// TIA Portal V16 export
// export: Created 2024-05-11T02:56:22.535184Z, ExportSetting WithDefaults, DisplayName Totally Integrated Automation Portal, DisplayVersion V16, DisplayName TIA Portal Version Control Interface, DisplayVersion V16, DisplayName TIA Portal Openness, DisplayVersion V16, DisplayName STEP 7 Professional, DisplayVersion V16, DisplayName STEP 7 Safety, DisplayVersion V16, DisplayName WinCC Professional, DisplayVersion V16
FUNCTION_BLOCK "K11_入口自动"   // FB11, LAD
{ S7_Optimized_Access := 'TRUE' }
VERSION : 0.1
// stored: AutoNumber false, IsIECCheckEnabled false, IsRetainMemResEnabled false, MemoryReserve 100, SetENOAutomatically false, UDAEnableTagReadback false
   VAR_TEMP
      EN_提升机上升指令 : Array[1..8] of Bool;
      EN_提升机下降指令 : Array[1..8] of Bool;
      EN_阻挡上升指令 : Array[1..8] of Bool;
      EN_阻挡下降指令 : Array[1..8] of Bool;
   END_VAR
   VAR_TEMP   // added for the SCL form of the ladder/FBD networks
      _w1 : Bool;
   END_VAR
BEGIN

REGION Network 1: @SN1=入口部
END_REGION

REGION Network 2: @选择分支
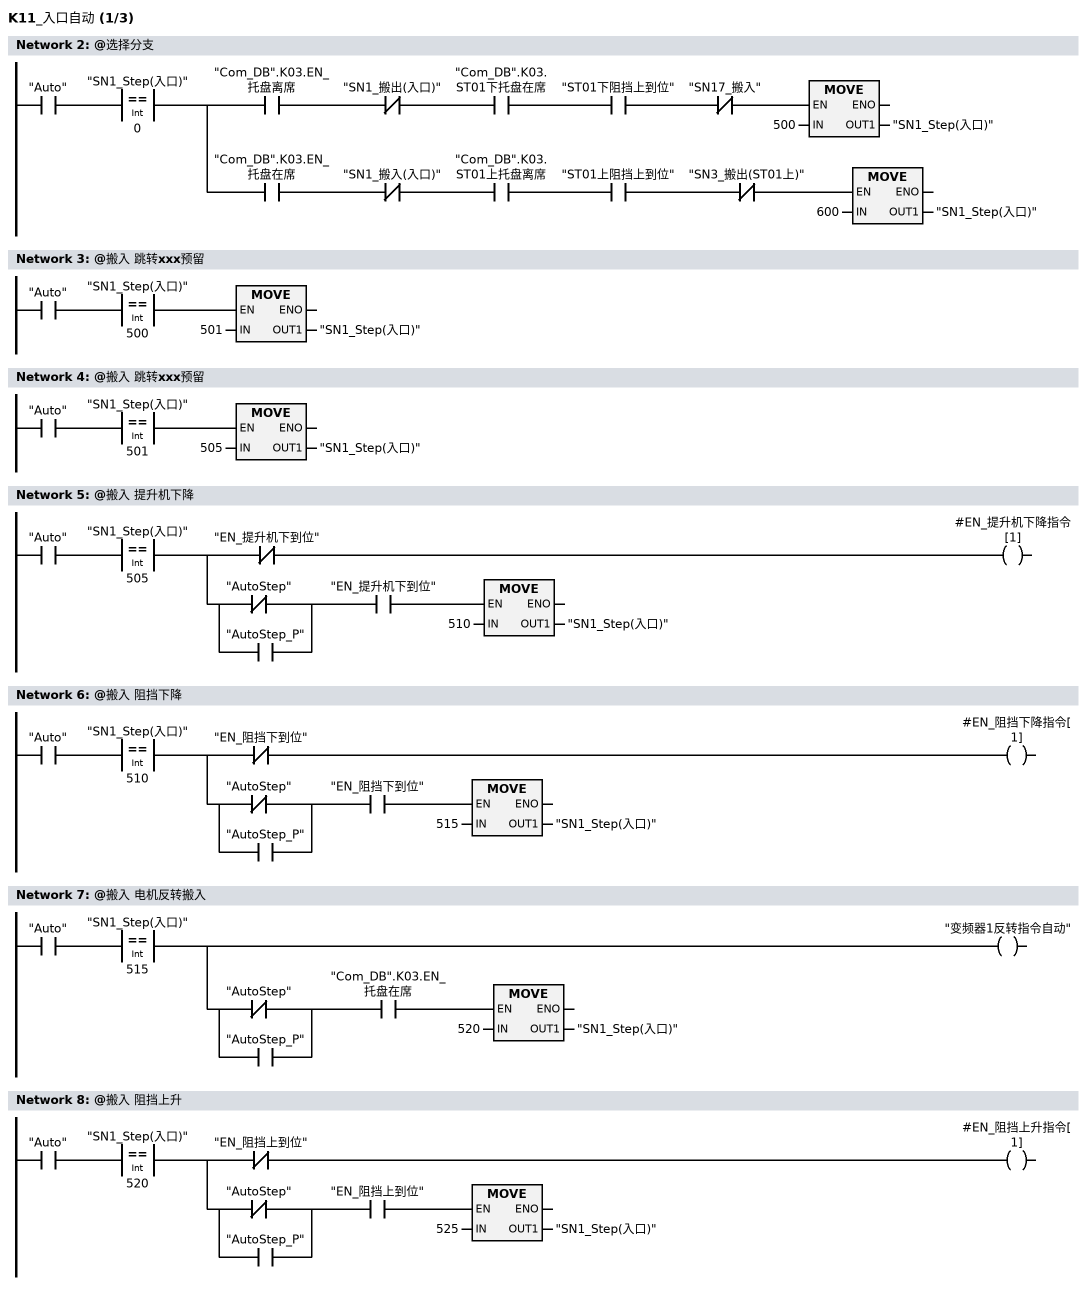
   RUNG wire#powerrail
      Contact( "Auto" )
      { S7_Templates := "SrcType := Int" } EQ_Contact(in1 := "SN1_Step(入口)", in2 := 0)
      wire#w1
      Contact( "Com_DB".K03.EN_托盘离席 )
      I_Contact( "SN1_搬出(入口)" )
      Contact( "Com_DB".K03.ST01下托盘在席 )
      Contact( "ST01下阻挡上到位" )
      I_Contact( "SN17_搬入" )
      Move(in := 500, out1 => "SN1_Step(入口)")
   END_RUNG
   RUNG wire#w1
      Contact( "Com_DB".K03.EN_托盘在席 )
      I_Contact( "SN1_搬入(入口)" )
      Contact( "Com_DB".K03.ST01上托盘离席 )
      Contact( "ST01上阻挡上到位" )
      I_Contact( "SN3_搬出(ST01上)" )
      Move(in := 600, out1 => "SN1_Step(入口)")
   END_RUNG
   // the same network as SCL:
   #_w1 := "Auto" AND ("SN1_Step(入口)" = 0);
   IF #_w1 AND "Com_DB".K03.EN_托盘离席 AND NOT "SN1_搬出(入口)" AND "Com_DB".K03.ST01下托盘在席 AND "ST01下阻挡上到位" AND NOT "SN17_搬入" THEN
       "SN1_Step(入口)" := 500;
   END_IF;
   IF #_w1 AND "Com_DB".K03.EN_托盘在席 AND NOT "SN1_搬入(入口)" AND "Com_DB".K03.ST01上托盘离席 AND "ST01上阻挡上到位" AND NOT "SN3_搬出(ST01上)" THEN
       "SN1_Step(入口)" := 600;
   END_IF;
END_REGION

REGION Network 3: @搬入 跳转xxx预留
   RUNG wire#powerrail
      Contact( "Auto" )
      { S7_Templates := "SrcType := Int" } EQ_Contact(in1 := "SN1_Step(入口)", in2 := 500)
      Move(in := 501, out1 => "SN1_Step(入口)")
   END_RUNG
   // the same network as SCL:
   IF "Auto" AND ("SN1_Step(入口)" = 500) THEN "SN1_Step(入口)" := 501; END_IF;
END_REGION

REGION Network 4: @搬入 跳转xxx预留
   RUNG wire#powerrail
      Contact( "Auto" )
      { S7_Templates := "SrcType := Int" } EQ_Contact(in1 := "SN1_Step(入口)", in2 := 501)
      Move(in := 505, out1 => "SN1_Step(入口)")
   END_RUNG
   // the same network as SCL:
   IF "Auto" AND ("SN1_Step(入口)" = 501) THEN "SN1_Step(入口)" := 505; END_IF;
END_REGION

REGION Network 5: @搬入 提升机下降
   RUNG wire#powerrail
      Contact( "Auto" )
      { S7_Templates := "SrcType := Int" } EQ_Contact(in1 := "SN1_Step(入口)", in2 := 505)
      wire#w1
      I_Contact( "EN_提升机下到位" )
      Coil( #EN_提升机下降指令[1] )
   END_RUNG
   RUNG wire#w1
      I_Contact( "AutoStep" )
      wire#w2
      Contact( "EN_提升机下到位" )
      Move(in := 510, out1 => "SN1_Step(入口)")
   END_RUNG
   RUNG wire#w1
      Contact( "AutoStep_P" )
   END_RUNG wire#w2
   // the same network as SCL:
   #_w1 := "Auto" AND ("SN1_Step(入口)" = 505);
   #EN_提升机下降指令[1] := #_w1 AND NOT "EN_提升机下到位";
   IF #_w1 AND (NOT "AutoStep" OR "AutoStep_P") AND "EN_提升机下到位" THEN "SN1_Step(入口)" := 510; END_IF;
END_REGION

REGION Network 6: @搬入 阻挡下降
   RUNG wire#powerrail
      Contact( "Auto" )
      { S7_Templates := "SrcType := Int" } EQ_Contact(in1 := "SN1_Step(入口)", in2 := 510)
      wire#w1
      I_Contact( "EN_阻挡下到位" )
      Coil( #EN_阻挡下降指令[1] )
   END_RUNG
   RUNG wire#w1
      I_Contact( "AutoStep" )
      wire#w2
      Contact( "EN_阻挡下到位" )
      Move(in := 515, out1 => "SN1_Step(入口)")
   END_RUNG
   RUNG wire#w1
      Contact( "AutoStep_P" )
   END_RUNG wire#w2
   // the same network as SCL:
   #_w1 := "Auto" AND ("SN1_Step(入口)" = 510);
   #EN_阻挡下降指令[1] := #_w1 AND NOT "EN_阻挡下到位";
   IF #_w1 AND (NOT "AutoStep" OR "AutoStep_P") AND "EN_阻挡下到位" THEN "SN1_Step(入口)" := 515; END_IF;
END_REGION

REGION Network 7: @搬入 电机反转搬入
   RUNG wire#powerrail
      Contact( "Auto" )
      { S7_Templates := "SrcType := Int" } EQ_Contact(in1 := "SN1_Step(入口)", in2 := 515)
      wire#w1
      Coil( "变频器1反转指令自动" )
   END_RUNG
   RUNG wire#w1
      I_Contact( "AutoStep" )
      wire#w2
      Contact( "Com_DB".K03.EN_托盘在席 )
      Move(in := 520, out1 => "SN1_Step(入口)")
   END_RUNG
   RUNG wire#w1
      Contact( "AutoStep_P" )
   END_RUNG wire#w2
   // the same network as SCL:
   "变频器1反转指令自动" := "Auto" AND ("SN1_Step(入口)" = 515);
   IF "变频器1反转指令自动" AND (NOT "AutoStep" OR "AutoStep_P") AND "Com_DB".K03.EN_托盘在席 THEN
       "SN1_Step(入口)" := 520;
   END_IF;
END_REGION

REGION Network 8: @搬入 阻挡上升
   RUNG wire#powerrail
      Contact( "Auto" )
      { S7_Templates := "SrcType := Int" } EQ_Contact(in1 := "SN1_Step(入口)", in2 := 520)
      wire#w1
      I_Contact( "EN_阻挡上到位" )
      Coil( #EN_阻挡上升指令[1] )
   END_RUNG
   RUNG wire#w1
      I_Contact( "AutoStep" )
      wire#w2
      Contact( "EN_阻挡上到位" )
      Move(in := 525, out1 => "SN1_Step(入口)")
   END_RUNG
   RUNG wire#w1
      Contact( "AutoStep_P" )
   END_RUNG wire#w2
   // the same network as SCL:
   #_w1 := "Auto" AND ("SN1_Step(入口)" = 520);
   #EN_阻挡上升指令[1] := #_w1 AND NOT "EN_阻挡上到位";
   IF #_w1 AND (NOT "AutoStep" OR "AutoStep_P") AND "EN_阻挡上到位" THEN "SN1_Step(入口)" := 525; END_IF;
END_REGION

REGION Network 9: @等搬入标志清除
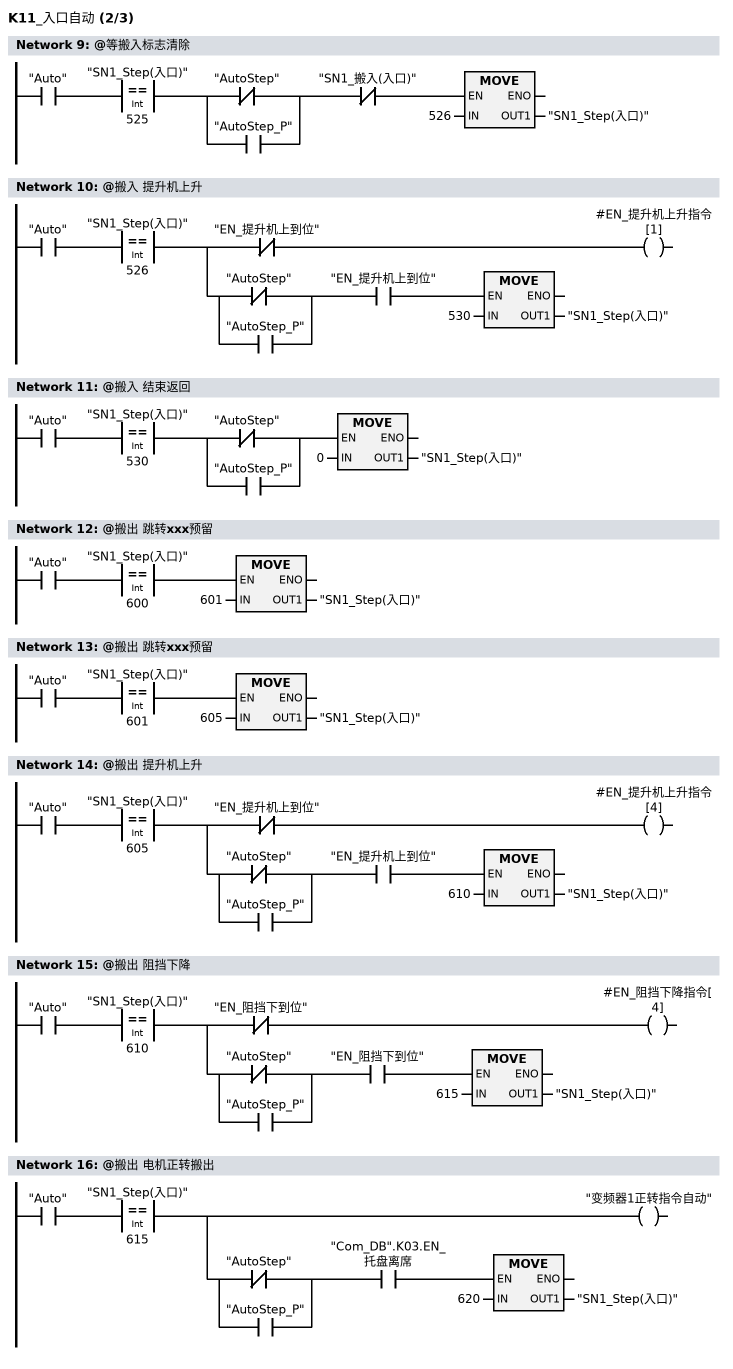
   RUNG wire#powerrail
      Contact( "Auto" )
      { S7_Templates := "SrcType := Int" } EQ_Contact(in1 := "SN1_Step(入口)", in2 := 525)
      wire#w1
      I_Contact( "AutoStep" )
      wire#w2
      I_Contact( "SN1_搬入(入口)" )
      Move(in := 526, out1 => "SN1_Step(入口)")
   END_RUNG
   RUNG wire#w1
      Contact( "AutoStep_P" )
   END_RUNG wire#w2
   // the same network as SCL:
   IF "Auto" AND ("SN1_Step(入口)" = 525) AND (NOT "AutoStep" OR "AutoStep_P") AND NOT "SN1_搬入(入口)" THEN
       "SN1_Step(入口)" := 526;
   END_IF;
END_REGION

REGION Network 10: @搬入 提升机上升
   RUNG wire#powerrail
      Contact( "Auto" )
      { S7_Templates := "SrcType := Int" } EQ_Contact(in1 := "SN1_Step(入口)", in2 := 526)
      wire#w1
      I_Contact( "EN_提升机上到位" )
      Coil( #EN_提升机上升指令[1] )
   END_RUNG
   RUNG wire#w1
      I_Contact( "AutoStep" )
      wire#w2
      Contact( "EN_提升机上到位" )
      Move(in := 530, out1 => "SN1_Step(入口)")
   END_RUNG
   RUNG wire#w1
      Contact( "AutoStep_P" )
   END_RUNG wire#w2
   // the same network as SCL:
   #_w1 := "Auto" AND ("SN1_Step(入口)" = 526);
   #EN_提升机上升指令[1] := #_w1 AND NOT "EN_提升机上到位";
   IF #_w1 AND (NOT "AutoStep" OR "AutoStep_P") AND "EN_提升机上到位" THEN "SN1_Step(入口)" := 530; END_IF;
END_REGION

REGION Network 11: @搬入 结束返回
   RUNG wire#powerrail
      Contact( "Auto" )
      { S7_Templates := "SrcType := Int" } EQ_Contact(in1 := "SN1_Step(入口)", in2 := 530)
      wire#w1
      I_Contact( "AutoStep" )
      wire#w2
      Move(in := 0, out1 => "SN1_Step(入口)")
   END_RUNG
   RUNG wire#w1
      Contact( "AutoStep_P" )
   END_RUNG wire#w2
   // the same network as SCL:
   IF "Auto" AND ("SN1_Step(入口)" = 530) AND (NOT "AutoStep" OR "AutoStep_P") THEN
       "SN1_Step(入口)" := 0;
   END_IF;
END_REGION

REGION Network 12: @搬出 跳转xxx预留
   RUNG wire#powerrail
      Contact( "Auto" )
      { S7_Templates := "SrcType := Int" } EQ_Contact(in1 := "SN1_Step(入口)", in2 := 600)
      Move(in := 601, out1 => "SN1_Step(入口)")
   END_RUNG
   // the same network as SCL:
   IF "Auto" AND ("SN1_Step(入口)" = 600) THEN "SN1_Step(入口)" := 601; END_IF;
END_REGION

REGION Network 13: @搬出 跳转xxx预留
   RUNG wire#powerrail
      Contact( "Auto" )
      { S7_Templates := "SrcType := Int" } EQ_Contact(in1 := "SN1_Step(入口)", in2 := 601)
      Move(in := 605, out1 => "SN1_Step(入口)")
   END_RUNG
   // the same network as SCL:
   IF "Auto" AND ("SN1_Step(入口)" = 601) THEN "SN1_Step(入口)" := 605; END_IF;
END_REGION

REGION Network 14: @搬出 提升机上升
   RUNG wire#powerrail
      Contact( "Auto" )
      { S7_Templates := "SrcType := Int" } EQ_Contact(in1 := "SN1_Step(入口)", in2 := 605)
      wire#w1
      I_Contact( "EN_提升机上到位" )
      Coil( #EN_提升机上升指令[4] )
   END_RUNG
   RUNG wire#w1
      I_Contact( "AutoStep" )
      wire#w2
      Contact( "EN_提升机上到位" )
      Move(in := 610, out1 => "SN1_Step(入口)")
   END_RUNG
   RUNG wire#w1
      Contact( "AutoStep_P" )
   END_RUNG wire#w2
   // the same network as SCL:
   #_w1 := "Auto" AND ("SN1_Step(入口)" = 605);
   #EN_提升机上升指令[4] := #_w1 AND NOT "EN_提升机上到位";
   IF #_w1 AND (NOT "AutoStep" OR "AutoStep_P") AND "EN_提升机上到位" THEN "SN1_Step(入口)" := 610; END_IF;
END_REGION

REGION Network 15: @搬出 阻挡下降
   RUNG wire#powerrail
      Contact( "Auto" )
      { S7_Templates := "SrcType := Int" } EQ_Contact(in1 := "SN1_Step(入口)", in2 := 610)
      wire#w1
      I_Contact( "EN_阻挡下到位" )
      Coil( #EN_阻挡下降指令[4] )
   END_RUNG
   RUNG wire#w1
      I_Contact( "AutoStep" )
      wire#w2
      Contact( "EN_阻挡下到位" )
      Move(in := 615, out1 => "SN1_Step(入口)")
   END_RUNG
   RUNG wire#w1
      Contact( "AutoStep_P" )
   END_RUNG wire#w2
   // the same network as SCL:
   #_w1 := "Auto" AND ("SN1_Step(入口)" = 610);
   #EN_阻挡下降指令[4] := #_w1 AND NOT "EN_阻挡下到位";
   IF #_w1 AND (NOT "AutoStep" OR "AutoStep_P") AND "EN_阻挡下到位" THEN "SN1_Step(入口)" := 615; END_IF;
END_REGION

REGION Network 16: @搬出 电机正转搬出
   RUNG wire#powerrail
      Contact( "Auto" )
      { S7_Templates := "SrcType := Int" } EQ_Contact(in1 := "SN1_Step(入口)", in2 := 615)
      wire#w1
      Coil( "变频器1正转指令自动" )
   END_RUNG
   RUNG wire#w1
      I_Contact( "AutoStep" )
      wire#w2
      Contact( "Com_DB".K03.EN_托盘离席 )
      Move(in := 620, out1 => "SN1_Step(入口)")
   END_RUNG
   RUNG wire#w1
      Contact( "AutoStep_P" )
   END_RUNG wire#w2
   // the same network as SCL:
   "变频器1正转指令自动" := "Auto" AND ("SN1_Step(入口)" = 615);
   IF "变频器1正转指令自动" AND (NOT "AutoStep" OR "AutoStep_P") AND "Com_DB".K03.EN_托盘离席 THEN
       "SN1_Step(入口)" := 620;
   END_IF;
END_REGION

REGION Network 17: @搬出 阻挡上升
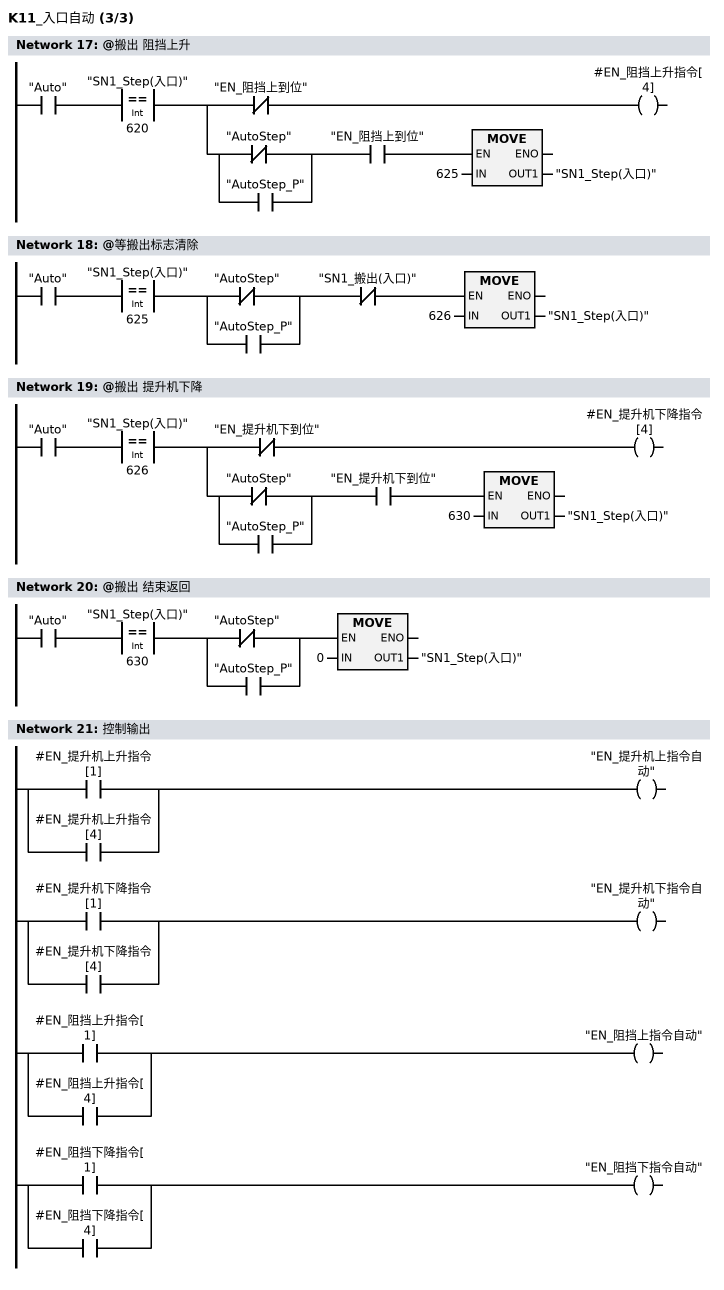
   RUNG wire#powerrail
      Contact( "Auto" )
      { S7_Templates := "SrcType := Int" } EQ_Contact(in1 := "SN1_Step(入口)", in2 := 620)
      wire#w1
      I_Contact( "EN_阻挡上到位" )
      Coil( #EN_阻挡上升指令[4] )
   END_RUNG
   RUNG wire#w1
      I_Contact( "AutoStep" )
      wire#w2
      Contact( "EN_阻挡上到位" )
      Move(in := 625, out1 => "SN1_Step(入口)")
   END_RUNG
   RUNG wire#w1
      Contact( "AutoStep_P" )
   END_RUNG wire#w2
   // the same network as SCL:
   #_w1 := "Auto" AND ("SN1_Step(入口)" = 620);
   #EN_阻挡上升指令[4] := #_w1 AND NOT "EN_阻挡上到位";
   IF #_w1 AND (NOT "AutoStep" OR "AutoStep_P") AND "EN_阻挡上到位" THEN "SN1_Step(入口)" := 625; END_IF;
END_REGION

REGION Network 18: @等搬出标志清除
   RUNG wire#powerrail
      Contact( "Auto" )
      { S7_Templates := "SrcType := Int" } EQ_Contact(in1 := "SN1_Step(入口)", in2 := 625)
      wire#w1
      I_Contact( "AutoStep" )
      wire#w2
      I_Contact( "SN1_搬出(入口)" )
      Move(in := 626, out1 => "SN1_Step(入口)")
   END_RUNG
   RUNG wire#w1
      Contact( "AutoStep_P" )
   END_RUNG wire#w2
   // the same network as SCL:
   IF "Auto" AND ("SN1_Step(入口)" = 625) AND (NOT "AutoStep" OR "AutoStep_P") AND NOT "SN1_搬出(入口)" THEN
       "SN1_Step(入口)" := 626;
   END_IF;
END_REGION

REGION Network 19: @搬出 提升机下降
   RUNG wire#powerrail
      Contact( "Auto" )
      { S7_Templates := "SrcType := Int" } EQ_Contact(in1 := "SN1_Step(入口)", in2 := 626)
      wire#w1
      I_Contact( "EN_提升机下到位" )
      Coil( #EN_提升机下降指令[4] )
   END_RUNG
   RUNG wire#w1
      I_Contact( "AutoStep" )
      wire#w2
      Contact( "EN_提升机下到位" )
      Move(in := 630, out1 => "SN1_Step(入口)")
   END_RUNG
   RUNG wire#w1
      Contact( "AutoStep_P" )
   END_RUNG wire#w2
   // the same network as SCL:
   #_w1 := "Auto" AND ("SN1_Step(入口)" = 626);
   #EN_提升机下降指令[4] := #_w1 AND NOT "EN_提升机下到位";
   IF #_w1 AND (NOT "AutoStep" OR "AutoStep_P") AND "EN_提升机下到位" THEN "SN1_Step(入口)" := 630; END_IF;
END_REGION

REGION Network 20: @搬出 结束返回
   RUNG wire#powerrail
      Contact( "Auto" )
      { S7_Templates := "SrcType := Int" } EQ_Contact(in1 := "SN1_Step(入口)", in2 := 630)
      wire#w1
      I_Contact( "AutoStep" )
      wire#w2
      Move(in := 0, out1 => "SN1_Step(入口)")
   END_RUNG
   RUNG wire#w1
      Contact( "AutoStep_P" )
   END_RUNG wire#w2
   // the same network as SCL:
   IF "Auto" AND ("SN1_Step(入口)" = 630) AND (NOT "AutoStep" OR "AutoStep_P") THEN
       "SN1_Step(入口)" := 0;
   END_IF;
END_REGION

REGION Network 21: 控制输出
   RUNG wire#powerrail
      Contact( #EN_提升机上升指令[1] )
      wire#w1
      Coil( "EN_提升机上指令自动" )
   END_RUNG
   RUNG wire#powerrail
      Contact( #EN_提升机上升指令[4] )
   END_RUNG wire#w1
   RUNG wire#powerrail
      Contact( #EN_提升机下降指令[1] )
      wire#w2
      Coil( "EN_提升机下指令自动" )
   END_RUNG
   RUNG wire#powerrail
      Contact( #EN_提升机下降指令[4] )
   END_RUNG wire#w2
   RUNG wire#powerrail
      Contact( #EN_阻挡上升指令[1] )
      wire#w3
      Coil( "EN_阻挡上指令自动" )
   END_RUNG
   RUNG wire#powerrail
      Contact( #EN_阻挡上升指令[4] )
   END_RUNG wire#w3
   RUNG wire#powerrail
      Contact( #EN_阻挡下降指令[1] )
      wire#w4
      Coil( "EN_阻挡下指令自动" )
   END_RUNG
   RUNG wire#powerrail
      Contact( #EN_阻挡下降指令[4] )
   END_RUNG wire#w4
   // the same network as SCL:
   "EN_提升机上指令自动" := #EN_提升机上升指令[1] OR #EN_提升机上升指令[4];
   "EN_提升机下指令自动" := #EN_提升机下降指令[1] OR #EN_提升机下降指令[4];
   "EN_阻挡上指令自动" := #EN_阻挡上升指令[1] OR #EN_阻挡上升指令[4];
   "EN_阻挡下指令自动" := #EN_阻挡下降指令[1] OR #EN_阻挡下降指令[4];
END_REGION
END_FUNCTION_BLOCK
